PROGRAM SecondUnit
VAR
	fbAlarm		: FB_Alarm;
	addAlarm	: BOOL;
END_VAR

IF addAlarm THEN
	fbAlarm.RaiseAlarm('This is Info from second unit');
	addAlarm := FALSE;
END_IF

END_PROGRAM

(* stored: Version 1.1.0.1, ProductVersion 3.1.4026.6
   POU SecondUnit: Id {cc68d63e-ecf6-4341-8ccd-b97ad0cbca79}, SpecialFunc None *)
